{attribute 'linkalways'} 
{attribute 'no_explicit_call' := 'This FB is a CLASS and must be accessed using methods or properties'}
{attribute 'enable_dynamic_creation'}
FUNCTION_BLOCK FINAL MUL_LREAL EXTENDS Node
VAR
	in1 : _LREAL(0.0);
	in2 : _LREAL(0.0);
	out : _LREAL(0.0);
END_VAR

METHOD PUBLIC Clone : I_Node
VAR
	pNode : POINTER TO MUL_LREAL;
END_VAR
pNode := __NEW(MUL_LREAL);
Clone := pNode^;
END_METHOD

METHOD FB_init : BOOL
VAR_INPUT
	bInitRetains : BOOL; // if TRUE, the retain variables are initialized (warm start / cold start)
	bInCopyCode : BOOL;  // if TRUE, the instance afterwards gets moved into the copy code (online change)
END_VAR
AddInput('in1',THIS^.in1);
AddInput('in2',THIS^.in2);
AddOutput('out', THIS^.out);
END_METHOD

METHOD PROTECTED OnExecute
VAR
END_VAR
out.Value := in1.Value * in2.Value;
END_METHOD

END_FUNCTION_BLOCK

(* stored: Version 1.1.0.1, ProductVersion 3.1.4024.15
   POU MUL_LREAL: Id {6e36f99d-3705-4893-ba0b-2c38ac44b210}, SpecialFunc None
   Folder Constructor: Id {c7bb7d5e-21d2-44fe-a28b-ced48bb0bc8d}
   Method Clone: Id {3ac25a91-9689-43b2-8ed9-538ef871f4f8}
   Method FB_init: Id {ab9269fd-16bf-4bfd-8a3c-58b75990b9a7}
   Method OnExecute: Id {32371114-582a-401f-aaba-32e973fe99b3} *)
